{attribute 'no_check' := ''}
//Sends Logbook entries handover by a LogbookPuplisher as SysLog messages to a SysLog Server 
//See wikipedia for more further inforamation about Syslog  
//based on TF6310 Tcp/Ip server 
FUNCTION_BLOCK LogbookSubSysLog IMPLEMENTS I_LogbookSubscriber
VAR CONSTANT
	MAX_BUFFER_LEVEL										:	INT := 85; //If buffer fill level reaches 85% Fb will appear as "busy2 to the LogBookPuplisher 
END_VAR

VAR CONSTANT 		
	MAX_SEND_STRING_SIZE									:	INT := 1024;
END_VAR
VAR_OUTPUT CONSTANT
{attribute 'displaymode':='binary'}
	OPTION_SYSLOG_WITH_FACILITY_SEVERITY_CODE				:	BYTE := 2#0000_0001;
{attribute 'displaymode':='binary'}
	OPTION_SYSLOG_WITH_RFC_5424_HEADER						:	BYTE := 2#0000_0010; //FALSE = RFC 3164 - Legacy Syslog / TRUE = RFC 5424 -> <134>1 2025-02-07T14:30:25.003Z server1 sshd 12345 ID47 [example@32473 iut="3" eventSource="ssh"] message 
{attribute 'displaymode':='binary'}
	OPTION_SYSLOG_WITH_CR									:	BYTE := 2#0000_0100; 
	{attribute 'displaymode':='binary'}
	OPTION_SYSLOG_WITH_LF									:	BYTE := 2#0000_1000; 
{attribute 'displaymode':='binary'}
//	OPTION_SYSLOG_WITH_TCP_MODE								:	BYTE := 2#0001_0000;
{attribute 'displaymode':='binary'}
	OPTION_SEND_STORED_MSG_WITH_DISABLE						: 	BYTE := 2#0010_0000; //Send stored messages if FB gets disabled to clear buffer
{attribute 'displaymode':='binary'}
	OPTION_ENABLE_BUFFER_ERROR								: 	BYTE := 2#0100_0000; //The FB changes to error state if the buffer was not emptied in time 	
{attribute 'displaymode':='binary'}
	OPTION_ENABLE_DEBUG										:	BYTE := 2#1000_0000; //Creates ADS log entries for conection events and errors
END_VAR
VAR_INPUT
	Enable													: 	BOOL;	//Enables sending new messages
	ResetTrig												:	BOOL;	//Ack error message
{attribute 'displaymode':='binary'}
	Options													:	BYTE := OPTION_SYSLOG_WITH_FACILITY_SEVERITY_CODE ; //option constants are alreay predefined, so they can accordingly be passed symbolically to the block
	SizeOfBuffer											:	UDINT := 2560; //Size of memory allocated from ads router memory pool by DoubleBuffer instance
	LocalHost	 											: 	T_IPv4Addr;  	//Local (client) address. String containing an (Ipv4) Internet Protocol dotted address. 
	LocalPort												:	UDINT := 515;	//Local (client) Internet Protocol (IP) port. (TCP Port = 1468) *)	
	RemoteHost	 											: 	T_IPv4Addr;  	//Remote (server) address. String containing an (Ipv4) Internet Protocol dotted address. 
	RemotePort												:	UDINT := 514;	//Remote (server) Internet Protocol (IP) port. (TCP Port = 1468) 
	Facility												:	BYTE := 16; 	//Default local 16
	Severity 												:	BYTE := 7; 		//0=Emergency/1=Alert/2=Critical/3=Error/4=Warning/5=Notice/6=Informational/7=Debug
	Tag														:	STRING(32) := ''; //Process name or local host by default
	LogPriorityLevel										:	UINT := 0; 		//0=All, correlates to EventClass priorities - see Para.EVENT_HANDLING_CONFIG priorities 1-3 
	PT_SendInterval											:	TIME := T#30S; //Messages will be send when buffer is filled or PT_SendInterval elapsed, T#0ms = off					
END_VAR                 				
VAR_OUTPUT              				        			
	Online													:	BOOL;		//TRUE if coonection is sucessful etablished
	hSocket													: 	T_HSOCKET ; //UDP Socket handle
	CntNoOfStoredMsgs										:	INT;
	TimeSendMsgs											:	TIME;
	Busy													: 	BOOL;  //Sending busy
	Error													: 	BOOL;	//Error occured
{attribute 'displaymode':='hex'}
	ErrorId													:	UDINT;	//See Beckhoff TF6310/ADS documentation for more information regarding error code
	ErrorFnc												:	STRING(20); //Error source 
	WinsockErrorId											:	E_WinsockError; //Winsocket error enum - see TF6310 documentation for further information
END_VAR
VAR
(* Memory ************************************************************)
	State													: 	INT := 0;
	SendCnt													:	UINT;
	StartTimeSendMsgs										:	TIME;
	SendErrorCnt											:	UINT;
	HeaderString											:	STRING;
	SendString												:	STRING(MAX_SEND_STRING_SIZE);
	SendStringLen											:	INT;
	_Severity												:	BYTE;
	LastMessageData											: 	LogbookData;
	LastEventClass											:	E_TcEventClass := TC2_SYSTEM.TCEVENTCLASS_NONE;
	
(* Trigger *****************************************************************)

(* Timer ******************************************************************)
	tonSendInterval											:	ton;
	
(* Blocks ***************************************************************)
	DblBuffer												:	DoubleBuffer;
	SocketClose												:	FB_SocketClose := (tTimeout := DEFAULT_ADS_TIMEOUT);
	SocketUdpCreate 										:	FB_SocketUdpCreate := (tTimeout := DEFAULT_ADS_TIMEOUT);
	SocketUdpSend											:	FB_SocketUdpSendTo := (tTimeout := T#10S);

(* Dummys *******************************************************************)
	i,j														:	INT;
END_VAR
(* 
Facality Description:
00 Kernel message
01 user-level messages
02 mail system
03 system daemons
04 security/authorization messages
05 messages generated internally by syslogd
06 line printer subsystem
07 network news subsystem
08 UUCP subsystem
09 clock daemon
10 security/authorization messages
11 FTP daemon
12 NTP subsystem
13 log audit
14 log alert
15 clock daemon
16 local10
17 local11
18 local12
19 local13
20 local14
21 local15
22 local16
23 local17

Severity Description:
0 Emergency
1 Alert
2 Critical
3 Error
4 Warning
5 Notice
6 Informational
7 Debug
*)

(* Logbook subscriber to send sys log messages via UDP 				*)
(********************************************************************)

(* Server connection ************************************************)
	CASE state OF
	0:
		IF Error
		THEN
			IF NOT Enable OR ResetTrig 
			THEN //Reset error
				Error										:= FALSE;
				ErrorId										:= 0;
				ErrorFnc									:= '';	
				WinsockErrorId								:= WSOK;			
			END_IF		
		ELSIF Online AND Enable
		THEN
			//Run interval
			tonSendInterval(IN := PT_SendInterval <> T#0MS AND CntNoOfStoredMsgs > 0 AND NOT DblBuffer.Empty, PT := PT_SendInterval);
			IF tonSendInterval.Q
			THEN
				tonSendInterval(IN := FALSE);
				DblBuffer.setReadyToRead(TRUE);
			END_IF
			
			IF DblBuffer.ReadyToRead //Buffer full or triggered by interval
			THEN
				CntNoOfStoredMsgs							:= 0;
				StartTimeSendMsgs							:= TIME();

				SocketUdpSend(
					sSrvNetId	:= , 
					hSocket		:= hSocket, 
					sRemoteHost	:= RemoteHost, 
					nRemotePort	:= RemotePort, 
					cbLen		:= DblBuffer.SizeOfDataToRead, 
					pSrc		:= DblBuffer.pDataToRead, 
					bExecute	:= TRUE, 
					tTimeout	:= , 
					bBusy		=> , 
					bError		=> , 
					nErrId		=> );
													
				state										:= 20;
			END_IF
		ELSIF Enable			
		THEN
			DblBuffer.SizeOfMemory							:= SizeOfBuffer;
			SocketUdpCreate(bExecute := FALSE);
			SocketClose(bExecute := FALSE);
			SocketUdpSend(bExecute := FALSE);
			Online											:= FALSE;
			Busy											:= TRUE;
			Error											:= FALSE;
			ErrorId											:= 0;
			ErrorFnc										:= '';	
			WinsockErrorId									:= WSOK;
			
			IF NOT SocketUdpCreate.bBusy
				AND NOT SocketClose.bBusy
				AND NOT SocketUdpSend.bBusy
			THEN
				tonSendInterval(IN := FALSE);
				SendCnt										:= 0;
				SendErrorCnt								:= 0;
				state										:= 10;
			END_IF	
		ELSE //Disabled
			IF hSocket.handle <> 0
			THEN //Close socket			
				IF NOT DblBuffer.Empty AND Options.5
				THEN //Write rest of buffer
					IF NOT DblBuffer.ReadyToRead THEN DblBuffer.setReadyToRead(TRUE); END_IF 
					CntNoOfStoredMsgs						:= 0;
					StartTimeSendMsgs						:= TIME();
					SocketUdpSend(
						sSrvNetId	:= , 
						hSocket		:= hSocket, 
						sRemoteHost	:= RemoteHost, 
						nRemotePort	:= RemotePort, 
						cbLen		:= DblBuffer.SizeOfDataToRead, 
						pSrc		:= DblBuffer.pDataToRead, 
						bExecute	:= TRUE, 
						tTimeout	:= , 
						bBusy		=> , 
						bError		=> , 
						nErrId		=> );
					State									:= 20;
				ELSE
					State									:= 30;
				END_IF			
			END_IF
		END_IF

	(* Create Socket *******************************************************)
	10: 
		SocketUdpCreate(
			sSrvNetId	:= , 
			sLocalHost	:= LocalHost, 
			nLocalPort	:= LocalPort, 
			bExecute	:= TRUE, 
			tTimeout	:= , 
			bBusy		=> , 
			bError		=> , 
			nErrId		=> , 
			hSocket		=> hSocket);
			
		IF NOT SocketUdpCreate.bBusy
		THEN
			IF SocketUdpCreate.bError
			THEN
				Error										:= TRUE;
				ErrorId										:= SocketUdpCreate.nErrId;
				ErrorFnc									:= 'SocketUdpCreate';
				WinsockErrorId								:= ADSERROR_TO_WSERROR(ErrorId);
				
				IF (Options AND OPTION_ENABLE_DEBUG) = 1
				THEN
					AdsLogError(CONCAT('LogbookClientSysLog | SocketUdpCreate %s | error id 16#', DWORD_TO_HEXSTR(TO_DWORD(ErrorID),4,FALSE)) ,HSOCKET_TO_STRING(SocketUdpCreate.hSocket));
				END_IF	

				state										:= 30;
			ELSE				
				hSocket.remoteAddr.sAddr					:= RemoteHost;
				hSocket.remoteAddr.nPort					:= RemotePort;
				
				IF (Options AND OPTION_ENABLE_DEBUG) = 1
				THEN
					AdsLogError(CONCAT('LogbookClientSysLog | SocketUdpCreate %s done', '') , HSOCKET_TO_STRING(SocketUdpCreate.hSocket));
				END_IF	
				
				Online 										:= TRUE;
				state										:= 0;
			END_IF		
			SocketUdpCreate(bExecute:= FALSE);
		END_IF		
		
	(* Send message ****************************************************)
	20:
		SocketUdpSend(
			sSrvNetId	:= , 
			hSocket		:= hSocket, 
			sRemoteHost	:= RemoteHost, 
			nRemotePort	:= RemotePort, 
			cbLen		:= DblBuffer.SizeOfDataToRead, 
			pSrc		:= DblBuffer.pDataToRead, 
			bExecute	:= TRUE, 
			tTimeout	:= , 
			bBusy		=> , 
			bError		=> , 
			nErrId		=> );
					
		IF NOT SocketUdpSend.bBusy
		THEN
			
			IF SocketUdpSend.bError
			THEN
				IF SendErrorCnt >= 3
				THEN
					Error									:= TRUE;
					ErrorId									:= SocketUdpSend.nErrId;
					ErrorFnc								:= 'SocketUdpSend';
					WinsockErrorId							:= ADSERROR_TO_WSERROR(ErrorId);
	
					IF (Options AND OPTION_ENABLE_DEBUG) = 1
					THEN
						AdsLogError(CONCAT('LogbookClientSysLog | SocketUdpSend %s | error id 16#', DWORD_TO_HEXSTR(TO_DWORD(ErrorID),4,FALSE)) ,HSOCKET_TO_STRING(SocketUdpCreate.hSocket));
					END_IF	
					
					State									:= 30; //Close socket
				ELSE //Try to send a second time
					SendErrorCnt							:= SendErrorCnt + 1;
				END_IF
			ELSE
				TimeSendMsgs								:= TIME() - StartTimeSendMsgs;		
				SendCnt										:= SendCnt + 1;		
				SendErrorCnt								:= 0;	
				DblBuffer.setReadyToRead(FALSE);
				State										:= 0;			
			END_IF 
				
			SocketUdpSend(bExecute := FALSE);
		END_IF
		
	(* Close socket ***********************************************)
	30:	
		SocketClose(
			sSrvNetId	:= , 
			hSocket		:= hSocket, 
			bExecute	:= hSocket.handle <> 0, 
			tTimeout	:= , 
			bBusy		=> , 
			bError		=> , 
			nErrId		=> );

		IF NOT SocketClose.bBusy
		THEN	
			IF SocketClose.bError 
			THEN
				IF NOT Error
				THEN
					Error									:= TRUE;
					ErrorId									:= SocketClose.nErrId;
					ErrorFnc								:= 'SocketUdpClose';
					WinsockErrorId							:= ADSERROR_TO_WSERROR(ErrorId);
				END_IF
				IF (Options AND OPTION_ENABLE_DEBUG) = 1
				THEN
					AdsLogError( CONCAT('LogbookClientSysLog | SocketClose %s | error id 16#', DWORD_TO_HEXSTR(TO_DWORD(ErrorID),4,FALSE)) ,HSOCKET_TO_STRING(SocketClose.hSocket));
				END_IF

				state										:= 0;				
			ELSE    
				IF (Options AND OPTION_ENABLE_DEBUG) = 1
				THEN
					AdsLogError( CONCAT('LogbookClientSysLog | SocketClose %s done', '') , HSOCKET_TO_STRING(SocketClose.hSocket));
				END_IF	
                      
				Online										:= FALSE;      
				hSocket.handle 								:= 0;          
				state										:= 0;
			END_IF		
			SocketClose(bExecute := FALSE);
		END_IF		
			
	END_CASE
	
(* Status *****************************************************************)
	Busy 													:= State <> 0 OR hSocket.handle <> 0 AND NOT Error;
	
(**************************************************************************)

METHOD PUBLIC FINAL addNewMessage : BOOL //Return value = TRUE if execution successful finished
VAR_IN_OUT
	data													:	LogbookData;
END_VAR
	IF Enable AND NOT Error
	THEN	
		LastMessageData									:= Data;
		LastEventClass.0								:= LastMessageData.Options.8;
		LastEventClass.1								:= LastMessageData.Options.9;
		LastEventClass.2								:= LastMessageData.Options.10;
		LastEventClass.3								:= LastMessageData.Options.11;
		
		CASE LastEventClass OF
		TC2_SYSTEM.TCEVENTCLASS_NONE		: _Severity		:= Severity; 		
		TC2_SYSTEM.TCEVENTCLASS_MESSAGE		: _Severity		:= 4;				
		TC2_SYSTEM.TCEVENTCLASS_HINT		: _Severity		:= 5;				
		TC2_SYSTEM.TCEVENTCLASS_STATEINFO	: _Severity		:= 6;				
		TC2_SYSTEM.TCEVENTCLASS_INSTRUCTION	: _Severity		:= 6;			 											
		TC2_SYSTEM.TCEVENTCLASS_WARNING		: _Severity		:= 4;	 			
		TC2_SYSTEM.TCEVENTCLASS_MAINTENANCE	: _Severity		:= 1;	 				 														
		TC2_SYSTEM.TCEVENTCLASS_ALARM		: _Severity		:= 0;	 			
		TC2_SYSTEM.TCEVENTCLASS_PARAMERROR	: _Severity		:= 3;	 			
		ELSE                                                                                     
			_Severity									:= 7;				
		END_CASE
	
		IF (LogPriorityLevel = 0 OR_ELSE GetEventClassPriority(LastEventClass) > LogPriorityLevel)
			AND_THEN CreateMsg(LastMessageData.Msg,LastMessageData.Timestamp ,_Severity)
		THEN
			IF DblBuffer.addData(ADR(SendString),TO_UDINT(SendStringLen)) <> S_OK
				AND Options.6
			THEN
				Error										:= TRUE;
				ErrorId										:= HRESULT_TO_ADSERROR(DblBuffer.hr);	
			ELSE
				CntNoOfStoredMsgs							:= CntNoOfStoredMsgs + 1;
			END_IF
		END_IF
		
		addNewMessage										:= NOT Error;	
	ELSE
		addNewMessage										:= FALSE;	
	END_IF
END_METHOD

METHOD PRIVATE FINAL createMsg : BOOL
VAR_IN_OUT
	MsgTxt													:	T_MaxString; (* 80/255 Zeichen *)
	MsgTime													:	TIMESTRUCT;	
	Severity												:	BYTE;
END_VAR                 									
VAR                     									
	TimeStamp												:	STRING(25);
	LenTxt													:	UDINT;
	LenHeader												:	UDINT;
END_VAR
IF NOT Options. 1 // OPTION_SYSLOG_WITH_RFC_5424_HEADER
THEN
	//Create Syslog msg RFC 5424 | <134>1 2025-02-07T14:30:25.003Z server1 sshd 12345 ID47 [example@32473 iut="3" eventSource="ssh"] message 
	IF (Options AND OPTION_SYSLOG_WITH_FACILITY_SEVERITY_CODE) <> 0 
	THEN 
		HeaderString 										:= REPLACE('<P>',BYTE_TO_STRING(SHL(FACILITY,3) OR (Severity AND BYTE#0000_0111)),1,2);	             										
	END_IF 
    
	//Sep 10 08:31:10
	CASE MsgTime.wMonth OF
	1: TimeStamp                                     		:= CONCAT(TimeStamp, ' Jan ');
	2: TimeStamp                                    		:= CONCAT(TimeStamp, ' Feb ');
	3: TimeStamp                                    		:= CONCAT(TimeStamp, ' Mar ');
	4: TimeStamp                                    		:= CONCAT(TimeStamp, ' Apr ');
	5: TimeStamp                                    		:= CONCAT(TimeStamp, ' May ');
	6: TimeStamp                                    		:= CONCAT(TimeStamp, ' Jun ');
	7: TimeStamp                                    		:= CONCAT(TimeStamp, ' Jul ');
	8: TimeStamp                                    		:= CONCAT(TimeStamp, ' Aug ');
	9: TimeStamp                                     		:= CONCAT(TimeStamp, ' Seb ');
	10:TimeStamp                                    		:= CONCAT(TimeStamp, ' Oct ');
	11:TimeStamp                                    		:= CONCAT(TimeStamp, ' Nov ');
	12:TimeStamp                                    		:= CONCAT(TimeStamp, ' Dec ');
	END_CASE
	
	TimeStamp                                         		:= CONCAT(TimeStamp,WORD_TO_STRING(MsgTime.wDay));
				
	IF MsgTime.wHour <10
	THEN
		TimeStamp 											:= Concat(TimeStamp,CONCAT(' 0',WORD_TO_STRING(MsgTime.wHour)));
	ELSE
		TimeStamp 											:= Concat(TimeStamp,CONCAT(' ',WORD_TO_STRING(MsgTime.wHour)));
	END_IF
	
	TimeStamp 												:= CONCAT(TimeStamp,':');
	
	IF MsgTime.wMinute < 10 
	THEN
		TimeStamp 											:= CONCAT(TimeStamp,CONCAT('0',WORD_TO_STRING(MsgTime.wMinute)));
	ELSE          										
		TimeStamp 											:= CONCAT(TimeStamp,WORD_TO_STRING(MsgTime.wMinute));
	END_IF
	
	TimeStamp 												:= CONCAT(TimeStamp,':');
	
	IF MsgTime.wSecond < 10 
	THEN
		TimeStamp 											:= CONCAT(TimeStamp,CONCAT('0',WORD_TO_STRING(MsgTime.wSecond)));
	ELSE
		TimeStamp 											:= CONCAT(TimeStamp,WORD_TO_STRING(MsgTime.wSecond));
	END_IF

	HeaderString 											:= CONCAT(HeaderString,TimeStamp);
	HeaderString 											:= CONCAT(HeaderString,' ');				
		
	(* ' host/sourcename eintragen (IP) *)
	HeaderString 											:= CONCAT(HeaderString, hSocket.localAddr.sAddr ); 
	
	(* Tag *)
	IF Len(Tag) > 0
	THEN
		HeaderString 										:= CONCAT(HeaderString,' '); 
		HeaderString										:= CONCAT(HeaderString,Tag);	
	END_IF
	HeaderString 											:= CONCAT(HeaderString,':'); 
	
ELSE //Create Syslog msg RFC 5424 | <134>1 2025-02-07T14:30:25.003Z server1 sshd 12345 ID47 [example@32473 iut="3" eventSource="ssh"] message 
	IF (Options AND OPTION_SYSLOG_WITH_FACILITY_SEVERITY_CODE) <> 0 
	THEN 
		HeaderString 										:= REPLACE('<P> 1 ',BYTE_TO_STRING(SHL(FACILITY,3) OR (Severity AND BYTE#0000_0111)),1,2);
		             										
	ELSE             										
		HeaderString 										:= '1 ';
	END_IF //1 is default version number

	
	//ISO 8601 timestamp, 2025-02-07T14:30:25.003 (local time)
	TimeStamp 											:= CONCAT(TimeStamp,WORD_TO_STRING(MsgTime.wYear));
				
	IF MsgTime.wMonth <10
	THEN
		TimeStamp 										:= Concat(TimeStamp,CONCAT('-0',WORD_TO_STRING(MsgTime.wMonth)));
	ELSE
		TimeStamp 										:= Concat(TimeStamp,CONCAT('-',WORD_TO_STRING(MsgTime.wMonth)));
	END_IF
	
	IF MsgTime.wDay <10
	THEN
		TimeStamp 										:= Concat(TimeStamp,CONCAT('-0',WORD_TO_STRING(MsgTime.wDay)));
	ELSE
		TimeStamp 										:= Concat(TimeStamp,CONCAT('-',WORD_TO_STRING(MsgTime.wDay)));
	END_IF
	
	
	IF MsgTime.wHour <10
	THEN
		TimeStamp 										:= Concat(TimeStamp,CONCAT('T0',WORD_TO_STRING(MsgTime.wHour)));
	ELSE
		TimeStamp 										:= Concat(TimeStamp,CONCAT('T',WORD_TO_STRING(MsgTime.wHour)));
	END_IF
	
	TimeStamp 											:= CONCAT(TimeStamp,':');
	
	IF MsgTime.wMinute < 10 
	THEN
		TimeStamp 										:= CONCAT(TimeStamp,CONCAT('0',WORD_TO_STRING(MsgTime.wMinute)));
	ELSE          										
		TimeStamp 										:= CONCAT(TimeStamp,WORD_TO_STRING(MsgTime.wMinute));
	END_IF
	
	TimeStamp 											:= CONCAT(TimeStamp,':');
	
	IF MsgTime.wSecond < 10 
	THEN
		TimeStamp 										:= CONCAT(TimeStamp,CONCAT('0',WORD_TO_STRING(MsgTime.wSecond)));
	ELSE
		TimeStamp 										:= CONCAT(TimeStamp,WORD_TO_STRING(MsgTime.wSecond));
	END_IF
	
	IF MsgTime.wMilliseconds < 10 
	THEN
		TimeStamp 										:= CONCAT(TimeStamp,CONCAT('.00',TO_STRING(MsgTime.wMilliseconds)));
	ELSIF MsgTime.wMilliseconds < 100
	THEN
		TimeStamp 										:= CONCAT(TimeStamp,CONCAT('.0',TO_STRING(MsgTime.wMilliseconds)));
	ELSE
		TimeStamp 										:= CONCAT(TimeStamp,CONCAT('.',TO_STRING(MsgTime.wMilliseconds)));
	END_IF
	
	HeaderString 										:= CONCAT(HeaderString,TimeStamp);
	HeaderString 										:= CONCAT(HeaderString,' ');				
		
	(* ' host/sourcename eintragen (IP) *)
	HeaderString 										:= CONCAT(HeaderString, hSocket.localAddr.sAddr ); 
	HeaderString 										:= CONCAT(HeaderString,' '); 
	
	(* Tag *)
	IF Len(Tag) > 0
	THEN
		HeaderString									:= CONCAT(HeaderString,Tag);
		HeaderString 									:= CONCAT(HeaderString,' '); 
	END_IF
	
	//Using "-" for "Process ID", "Message ID" and "[Data Structure]", as not applied
	HeaderString 										:= CONCAT(HeaderString,'- - - '); 
	
END_IF

	IF Options.2 
	THEN //CR
		MsgTxt											:= CONCAT(MsgTxt,'$r');
	END_IF
	
	IF Options.3 
	THEN //LF
		MsgTxt											:= CONCAT(MsgTxt,'$n');
	END_IF
	
	(* Msg *)
	SendString											:= HeaderString;
	SendStringLen										:= MIN(MAX_SEND_STRING_SIZE,(LEN(HeaderString) + Len(MsgTxt)));
	MEMCPY(ADR(SendString) + LEN(HeaderString), ADR(MsgTxt) , INT_TO_UDINT(LEn(MsgTxt)));
	SendString[SendStringLen] 							:= 0; //Terminate string
	
	CreateMsg											:= TRUE;
END_METHOD

{attribute 'monitoring' := 'call'}
PROPERTY PUBLIC isBusy : BOOL
GET
isBusy											:= DblBuffer.Full and Enable and not Error and DblBuffer.fillLevel >= MAX_BUFFER_LEVEL;
END_GET
END_PROPERTY

PROPERTY PUBLIC optAdd_CR : BOOL
GET
optAdd_CR := Options.2;
END_GET
SET
OPtions.2 := optAdd_CR;
END_SET
END_PROPERTY

PROPERTY PUBLIC optAdd_LF : BOOL
GET
optAdd_LF := Options.3;
END_GET
SET
Options.3 := optAdd_LF;
END_SET
END_PROPERTY

PROPERTY PUBLIC optEnabelDebugMode : BOOL
GET
optEnabelDebugMode := Options.7;
END_GET
SET
Options.7 := optEnabelDebugMode;
END_SET
END_PROPERTY

PROPERTY PUBLIC optEnableBufferError : BOOL
GET
optEnableBufferError := Options.6;
END_GET
SET
OPtions.6				:= optEnableBufferError;
END_SET
END_PROPERTY

PROPERTY PUBLIC optEnableFacilitySeverityCode : BOOL
GET
 optEnableFacilitySeverityCode := Options.0;
END_GET
SET
Options.0 := optEnableFacilitySeverityCode;
END_SET
END_PROPERTY

PROPERTY PUBLIC optEnableRFCHeader : BOOL
GET
optEnableRFCHeader := Options.1;
END_GET
SET
Options.1 := optEnableRFCHeader;
END_SET
END_PROPERTY

PROPERTY PUBLIC optSendMsgIfDisabled : BOOL
GET
optSendMsgIfDisabled := Options.5;
END_GET
SET
Options.5 := optSendMsgIfDisabled;
END_SET
END_PROPERTY

END_FUNCTION_BLOCK

(* stored: Version 1.1.0.1, ProductVersion 3.1.4024.13
   POU LogbookSubSysLog: Id {3b5ef261-afb1-4a5d-8cbb-5277a8c3f860}, SpecialFunc None
   Folder methods: Id {158d0774-089b-426d-9f7e-6833e240612d}
   Folder properties: Id {a90624a5-4cbb-442d-abb6-09c5f05b5a37}
   Folder options: Id {0cbaab93-28db-40aa-a1e7-913a4081737c}
   Method addNewMessage: Id {3bfbbec5-b586-4f55-9ddd-111f28a63046}
   Method createMsg: Id {aa74bb2f-5045-40cf-a7ae-83d0020ac346}
   Property isBusy: Id {e67702ae-1ac7-4830-b5d5-6fa289354da8}
   Get Get: Id {c87e46ff-cf63-464d-8373-9fdadd417f4a}
   Property optAdd_CR: Id {48adad1c-b04f-42f7-beeb-45fb02b12183}
   Get Get: Id {d5b90a0a-cc22-43e1-9d23-b3958558e37a}
   Set Set: Id {48400278-58de-4d2f-bd32-697c2c91d436}
   Property optAdd_LF: Id {b4c298da-5f33-470e-b7bf-7c7485c0a5c5}
   Get Get: Id {8ef9ef16-c1e6-4dbe-8b30-1d8282b786f1}
   Set Set: Id {62a6c846-626f-43e7-be3a-3568f8118a80}
   Property optEnabelDebugMode: Id {da68f2b2-32a2-4b13-8aad-e8cb39c417f3}
   Get Get: Id {1f7ea493-06ea-4f32-ba8f-5f925b9ea86a}
   Set Set: Id {2e5aea28-87da-43b7-bf04-3a8d38e594ca}
   Property optEnableBufferError: Id {b3c97c57-5dee-4e5e-b72d-933944fa6411}
   Get Get: Id {8256b78f-4e92-43a0-b104-b787c2d34599}
   Set Set: Id {6dc29065-1d14-4fe0-bd47-082001de5f49}
   Property optEnableFacilitySeverityCode: Id {294d44f3-64b4-47f6-8c39-593eb4969039}
   Get Get: Id {31eae8cb-eea9-4e98-a2e0-d378477d9d8e}
   Set Set: Id {efa182dc-1072-4c31-b41e-8b25028e7c05}
   Property optEnableRFCHeader: Id {ef99c11f-46ce-49b9-9c1b-818275b2a848}
   Get Get: Id {7946e1e3-8716-4988-9133-ab2e587bc603}
   Set Set: Id {cfdf19d7-d971-46b1-92b0-6984b7f3e5da}
   Property optSendMsgIfDisabled: Id {c59d3f7e-f031-45b0-81e5-6c5827029fd5}
   Get Get: Id {4d3ec294-06ec-44d6-bb15-e88bc8f5b58f}
   Set Set: Id {3254600d-7b2a-424a-afa7-fe737f6db0dd} *)
